PROGRAM MAIN
VAR
END_VAR

END_PROGRAM

(* stored: Version 1.1.0.1
   POU MAIN: Id {9dc25a2f-1af6-4ed0-81f3-885d9f4b74a7} *)
